# EPICS substitutions: epics/m-epics-eemcu/eemcuApp/Db/Sim8-extra-m2.substitutions
file "eemcu-extra.template"
{
pattern
{P,      M,    R,   PORT, ADDR, PREC, HOMEPROC}
{IOC:,   m2, m2-,   MCU1,    2, 3,    3}
}
